(* PLC project PLC_ODOT.project, CODESYS CODESYS V3.5 SP19 *)
(* stored: creationDateTime 2026-01-26T16:59:15.5899917, modificationDateTime 2026-01-26T16:51:59.9229809 *)

FUNCTION_BLOCK FbFilterA
  VAR_INPUT
    In : REAL := 0;  (* Входной сигнал до фильтрации. *)
    Tf : REAL := 1;  (* Постоянная времени фильтра [с]. *)
    Ts : REAL := 0.1;  (* Шаг дискретизации по времени [с]. *)
  END_VAR
  VAR_OUTPUT
    Out : REAL := 0;  (* Выходной сигнал после фильтрации. *)
  END_VAR
  VAR_TEMP
    Tmp : REAL;  (* Временная переменная вход интегратора. *)
  END_VAR

            //      DbFilterA
//    +-----------+
//    | FbFilterA |
// ->-|In      Out|->-
//   -|Tf         |
//   -|Ts         |
//    +-----------+

//W(s) = 1 / (1 + Tf * s) при Ts->0.
IF (Tf <= 0.0) THEN
Out := In;
ELSE
Tmp := (In - Out) / Tf;
Out := Out + Tmp * Ts;
END_IF;

// Внутренняя схема фильтра.
//
//          Вычитание   Деление      Интегрирование
//            +---+     +------+     +----------+
// In ----->--| + |     |   1  | Tmp |  Ts * z  |
//            |   |-->--| ---- |-->--| -------- |--+-->-- Out
//      +-->--| - |     |  Tf  |     |   z - 1  |  |
//      |     +---+     +------+     +----------+  |
//      |                                          |
//      +------------------------------------------+

// Условное графическое обозначение (приближенное).
//
//    +--------------+
//    |      1       |
// ->-| ------------ |->-
//    |  Tf * s + 1  |
//    +--------------+

// Электрическая схема фильтра.
//
//         R                  
// +    +-----+              +
// o----|     |----o---------o
//      +-----+    |          
//                 | C        
//               -----        
// U In          -----   U Out
//                 |          
// -               |         -
// o---------------o---------o
// Tf = R * C ([с] = [Ом] * [Ф])

// Временная характеристика.
//
// ^ Out
// |
// 1         *** Y(t) = 1 - exp(-(t/Tf))
// |      *     
// |    *       
// |  *         
// | *          
// 0---------------> t[s]
//
// ^ In
// |
// 1************ X(t) = 1
// |            
// |            
// |            
// |            
// 0---------------> t[s]

//  +---------+
//  | GNU GPL |
//  +---------+
//  |
//  |
//  .= .-_-. =.
// ((_/)o o(\_))
//  `-'(. .)`-'
//  |/| \_/ |\
//  ( |     | )
//  /"\_____/"\
//  \__)   (__/
// @COPYLEFT ALL WRONGS RESERVED :)
// Author: VA
// Contacts: DIY.PLC.314@gmail.com
// License: GNU GPL v2
//
// https://www.youtube.com/@DIY_PLC
// https://github.com/DIYPLC

          
END_FUNCTION_BLOCK
